FUNCTION_BLOCK CHOICE_TBL (* Table CHOICE input *)
  (* Standard: 61499-1; Classification: GUI *)
  (* Version 0.0, 2000-04-07, JHC, Rockwell Automation *)
  (* Compiler header: package fb.rt.hmi; import fb.rt.math.*; *)
  (* Compiler Java IBM VisualAge 3.0 *)
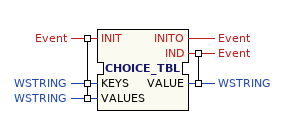
  EVENT_INPUT
    INIT WITH KEYS, VALUES; (* Table Initialization *)
  END_EVENT
  EVENT_OUTPUT
    INITO; (* Initialization Confirm *)
    IND WITH VALUE; (* New Choice *)
  END_EVENT
  VAR_INPUT
    KEYS : WSTRING; (* Comma-separated List of Keys *)
    VALUES : WSTRING; (* Comma-separated List of Values *)
  END_VAR
  VAR_OUTPUT
    VALUE : WSTRING; (* Value Corresponding to Chosen Key *)
  END_VAR
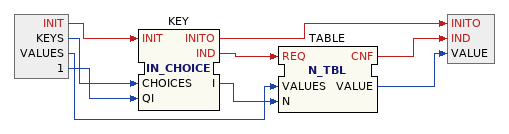
  FBS
    KEY : IN_CHOICE;
    TABLE : N_TBL;
  END_FBS
  EVENT_CONNECTIONS
    INIT TO KEY.INIT;
    KEY.INITO TO INITO;
    KEY.IND TO TABLE.REQ;
    TABLE.CNF TO IND;
  END_CONNECTIONS
  DATA_CONNECTIONS
    KEYS TO KEY.CHOICES;
    VALUES TO TABLE.VALUES;
    KEY.I TO TABLE.N;
    TABLE.VALUE TO VALUE;
    1 TO KEY.QI;
  END_CONNECTIONS
END_FUNCTION_BLOCK
